TYPE ST_ClampStationParCmd :
STRUCT
    Reserved : BOOL;
END_STRUCT
END_TYPE

(* stored: Version 1.1.0.1, ProductVersion 3.1.4024.12
   DUT ST_ClampStationParCmd: Id {a4f57e35-c9ed-424d-884e-282f9f83bace} *)
